// TIA Portal V18 export
DATA_BLOCK "DB_PARAMETERS_TEACH"   // DB7
{ S7_Optimized_Access := 'TRUE' }
// stored: MemoryReserve 100
   VAR
      HMI_PAGE_CONTROL : Struct
         TEACH_MODE_ACTIVE : Bool := FALSE;
         READ_CHOOSED_RECIPE : Bool := FALSE;
         NUMBER_OF_RECIPE : USInt := 1;
         SAVE_CHANGES_IN_RECIPE : Bool := FALSE;
         Use_recipe_Nbr : USInt := 1;
         Use_recipe_trigger : Bool := false;
         Speeds : Struct
            Glue_IAI : Struct
               X : Int := 10;
               Y : Int := 10;
               Z : Int := 10;
            END_STRUCT;
            A1_table : Int := 500;
            A2_table : Int := 500;
            Shaft_rotation : Int := 500;
            Glue_rotation : Int := 500;
         END_STRUCT;
         Go_to_pos : Struct
            Glue_IAI : Struct
               X : Real;
               Y : Real;
               Z : Real;
            END_STRUCT;
            A1_table : Int;
            A2_table : Int;
            Shaft_rotation : Int;
            Glue_rotation : Int;
         END_STRUCT;
         Go_to_pos_TRIGGER : Struct
            Glue_IAI : Struct
               X : Bool := FALSE;
               Y : Bool := FALSE;
               Z : Bool := FALSE;
            END_STRUCT;
            A1_table : Bool := FALSE;
            A2_table : Bool := FALSE;
            Shaft_rotation : Bool := FALSE;
            Glue_rotation : Bool := FALSE;
         END_STRUCT;
      END_STRUCT;
      "TEACH SCREEN VALUES" : "UDT_OP10_Recipe_type";
   END_VAR
BEGIN
END_DATA_BLOCK
